Universal Robots URScript: v2.1ross.script

def v21ross():
  set_gravity([0.0, 0.0, 9.82])
  set_safety_mode_transition_hardness(0)
  set_tool_voltage(24)
  set_standard_analog_input_domain(0, 1)
  set_standard_analog_input_domain(1, 1)
  set_tool_analog_input_domain(0, 0)
  set_tool_analog_input_domain(1, 0)
  set_analog_outputdomain(0, 1)
  set_analog_outputdomain(1, 0)
  set_input_actions_to_default()
  set_tcp(p[0.0,0.0,0.18,0.0,3.14,0.0])
  set_payload(0.71, [0.0, 0.0, 0.275])
  step_count_50fda1c7_9b45_4d17_a144_ef9c53115f70 = 0.0
  thread Step_Counter_Thread_b07ae2ea_29d2_4196_91c5_4a2053767ce3():
    while (True):
      step_count_50fda1c7_9b45_4d17_a144_ef9c53115f70 = step_count_50fda1c7_9b45_4d17_a144_ef9c53115f70 + 1.0
      sync()
    end
  end
  run Step_Counter_Thread_b07ae2ea_29d2_4196_91c5_4a2053767ce3()
  global plane=[0, 0, 0, 0, 0, 0]
  global free=1
  global Gaveteiro_plane=p[-0.18391406007170819,-0.6890912013208738,-0.3091053148893457,-3.136624244641354,-0.07450754164245207,-0.012062489851684073]
  global Plane_var=p[0.0455072287759728,0.5532633607914713,-0.12009520789912541,0.02088120484419274,0.010016746118093,-0.02458726325044075]
  global PlanoMesaAula9=p[0.4316603038800538,-0.4176154966413232,-0.22708615915239258,0.0011409468517281232,-0.0021558803218785405,-3.3834622272085614E-4]
  global Plano_BotRoss=p[-0.05323872750160344,0.3963224432691249,-0.20848789913917903,0.041759501527263314,0.014917504040608983,0.11867115612734513]
  global Plano_mesa_gio=p[0.5722610509435332,-0.40820095277647794,-0.22787514661355984,0.004980319709535583,-0.010045557410892312,0.003475544605146006]
  global socketIP=p[0.7942382577522773,-0.05274490106868765,0.28953087333027294,-1.2101977474418126,-1.2112243285351472,1.2072853144995164]
  global xadrez=p[0.07245008429201542,0.7162309814300137,-0.2492325678677777,0.021240702277102536,0.009909632298596038,-2.9870755951116497]
  global xadrez2=p[-0.24762135118614845,0.3378039779312413,-0.2536888643835707,0.03547999981100722,-0.008259935265332035,0.09585250855875074]
  rtde_set_watchdog("speed_slider_mask", 10.0, "ignore")
  $ 1 "BeforeStart"
  $ 2 "Socket≔socket_open('10.103.16.11',20000)"
  global Socket=socket_open("10.103.16.11",20000)
  $ 3 "Num_points≔socket_read_ascii_float(1)"
  global Num_points=socket_read_ascii_float(1)
  while (True):
    $ 4 "Robot Program"
    $ 5 "Loop Socket≟ False "
    while (Socket ==   False  ):
      $ 6 "Socket≔socket_open('10.103.16.11',20000)"
      global Socket=socket_open("10.103.16.11",20000)
    end
    $ 7 "Num_points≔socket_read_ascii_float(1)"
    global Num_points=socket_read_ascii_float(1)
    $ 8 "N≔Num_points[1]"
    global N=Num_points[1]
    $ 9 "X≔socket_read_ascii_float(N)"
    global X=socket_read_ascii_float(N)
    $ 10 "Y≔socket_read_ascii_float(N)"
    global Y=socket_read_ascii_float(N)
    $ 11 "Z≔socket_read_ascii_float(N)"
    global Z=socket_read_ascii_float(N)
    $ 13 "count≔1"
    global count=1
    $ 14 "Loop count≤N"
    while (count <= N):
      $ 15 "move2pose≔p[X[count]/1000,Y[count]/1000,Z[count]/1000,0,0,0]"
      global move2pose=p[X[count]/1000,Y[count]/1000,Z[count]/1000,0,0,0]
      $ 16 "MoveL"
      $ 17 "move2pose" "breakAfter"
      movel(pose_trans(Plano_BotRoss, move2pose), a=0.6, v=0.2)
      $ 19 "count≔count+1"
      global count=count+1
    end
  end
end
